{attribute 'no_explicit_call' := 'This FB is a CLASS and must be accessed using methods or properties'}
{attribute 'enable_dynamic_creation'}
{attribute 'hide_all_locals'}
FUNCTION_BLOCK FB_DynamicArray
VAR
	buffer : FB_JsonDynDomParser;
	root : sJsonValue;
END_VAR

PROPERTY PRIVATE _Array : sJsonValue
GET
IF root <> 0 THEN
	_Array := root;
ELSE
	root := buffer.NewDocument();
	_Array := buffer.SetArray(root,0);
END_IF
END_GET
END_PROPERTY

METHOD PUBLIC AddLast : BOOL
VAR_INPUT
	Value : ANY;
END_VAR
AddLast := buffer.PushbackBase64Value(v:= _Array, p := Value.pValue,n := Value.diSize) <> 0;
END_METHOD

METHOD PUBLIC AddStringLast : BOOL
VAR_INPUT
	Value : ANY_STRING;
END_VAR
AddStringLast := buffer.PushbackBase64Value(v:= _Array, p := Value.pValue,n := TO_DINT(LEN2(Value.pValue)+ 1)) <> 0;
END_METHOD

METHOD PUBLIC Clear : BOOL
VAR
	_arrayElement : SJsonAIterator;
END_VAR
_arrayElement := buffer.ArrayBegin(_array);
IF _arrayElement <> 0 THEN
	Clear := buffer.ClearArray(v := _array,i := _arrayElement);
END_IF
END_METHOD

METHOD PUBLIC CopyArrayString : BOOL
VAR_IN_OUT CONSTANT
  	pDoc : STRING; 
END_VAR
VAR_INPUT
	nDoc : UDINT;
END_VAR
CopyArrayString := buffer.copyjson(v:= _Array, pDoc:= pDoc,nDoc := nDoc) <> 0;
END_METHOD

PROPERTY PUBLIC Count : UDINT
GET
Count := buffer.GetArraySize(_array);
END_GET
END_PROPERTY

PROPERTY PUBLIC FirstIndex : UDINT
GET
FirstIndex := 0;
END_GET
END_PROPERTY

PROPERTY PUBLIC LastIndex : UDINT
GET
IF Count = 0 THEN
	LastIndex := 0;
ELSE 
	LastIndex := Count - 1;
END_IF
END_GET
END_PROPERTY

METHOD PUBLIC RemoveFirst : BOOL
VAR
	_arrayElement : SJsonAIterator;
END_VAR
RemoveFirst := TryDeleteIndex(0);
END_METHOD

METHOD PUBLIC RemoveLast: BOOL
VAR
	_arrayElement : SJsonAIterator;
END_VAR
RemoveLast := TryDeleteIndex(LastIndex);
END_METHOD

METHOD PUBLIC TryDeleteIndex : BOOL
VAR_INPUT
	Index : UDINT;
END_VAR
VAR
	_arrayElement : SJsonAIterator;
END_VAR
_arrayElement := buffer.GetArrayValueByIdx(_Array, Index);
IF _arrayElement <> 0 THEN
	TryDeleteIndex := buffer.RemoveArray(v := _array,i := _arrayElement);
END_IF
END_METHOD

METHOD PUBLIC TryGetIndex : BOOL;
VAR_INPUT
	Index : UDINT;
	Destination : ANY;
END_VAR
TryGetIndex := buffer.GetBase64(v:=  buffer.GetArrayValueByIdx(_Array, Index),p := Destination.pValue, n:= Destination.diSize) <> 0;
END_METHOD

METHOD PUBLIC TryGetIndexTo : BOOL;
VAR_INPUT
	Index : UDINT;
	Destination : PVOID;
	DestinationSize : UDINT;
END_VAR
VAR
	_arrayElement : SJsonAIterator;
END_VAR
_arrayElement := buffer.GetArrayValueByIdx(_Array, Index);
IF _arrayElement <> 0 THEN
	TryGetIndexTo := buffer.GetBase64(v:= _arrayElement,p := Destination, n:= TO_DINT(DestinationSize)) <> 0;
END_IF
END_METHOD

METHOD PUBLIC TrySetIndex : BOOL
VAR_INPUT
	Index : UDINT;
	Value : ANY;
END_VAR
TrySetIndex := buffer.SetBase64(v:= buffer.GetArrayValueByIdx(_Array, Index),p := Value.pValue, n:= Value.diSize) <> 0;
END_METHOD

METHOD PUBLIC TrySetIndexTo : BOOL
VAR_INPUT
	Index : UDINT;
	Value : PVOID;
	ValueSize : UDINT;
END_VAR
VAR
	_arrayElement : SJsonAIterator;
END_VAR
_arrayElement := buffer.GetArrayValueByIdx(_Array, Index);
IF _arrayElement <> 0 THEN
	TrySetIndexTo := buffer.SetBase64(v:= _arrayElement,p := Value, n:= TO_DINT(ValueSize)) <> 0;
END_IF
END_METHOD

END_FUNCTION_BLOCK

(* stored: Version 1.1.0.1, ProductVersion 3.1.4024.12
   POU FB_DynamicArray: Id {1195ebad-f841-400e-9a73-9ed4923ff5ec}, SpecialFunc None
   Folder Private: Id {49466fda-f5e0-4ad7-b43a-0352687a0c9c}
   Property _Array: Id {7d52bff1-ae95-47c5-a3a6-f6a3c9ae2414}
   Get Get: Id {9b7aeaa8-6d0e-42e1-979f-220b44e2b3f8}
   Method AddLast: Id {c8a7e319-c35e-429c-93ba-1476380fe1dd}
   Method AddStringLast: Id {aa636f09-5b04-45bc-9bba-0b69ecbe8c47}
   Method Clear: Id {3729fa69-f5b0-44e7-83e0-cc5cbbe6f4c8}
   Method CopyArrayString: Id {9aea8499-b935-4a78-9cc9-344b7bef6e5c}
   Property Count: Id {cb41e7a9-313d-4b1e-bf36-f46b8963868e}
   Get Get: Id {dcbd6a1c-3944-46e8-9299-a1af2bca0c96}
   Property FirstIndex: Id {9a033c19-af18-451c-b0af-245999fa4197}
   Get Get: Id {63187c88-c9ec-4da2-a631-3e9d6cd8d435}
   Property LastIndex: Id {edb01bc9-cfe2-4196-b5ac-84b13bdcb4b5}
   Get Get: Id {e7a0207e-d433-4a9e-aa23-7a581f253aa9}
   Method RemoveFirst: Id {7e0230e0-0608-417f-95e6-f49abdba3f67}
   Method RemoveLast: Id {27237050-c8a0-43fa-8f3d-0f08d2838c8c}
   Method TryDeleteIndex: Id {7cd6dc9a-7bd8-4ed1-ba00-31d671654630}
   Method TryGetIndex: Id {00128fb3-0888-4680-baae-fe94bc38c29b}
   Method TryGetIndexTo: Id {1412ae45-9668-4dda-b44d-6048d41a0a8b}
   Method TrySetIndex: Id {5ccebf41-1520-4351-9dd1-6cb87d270b62}
   Method TrySetIndexTo: Id {5b14ca33-060c-429e-8e33-05638c5831c8} *)
